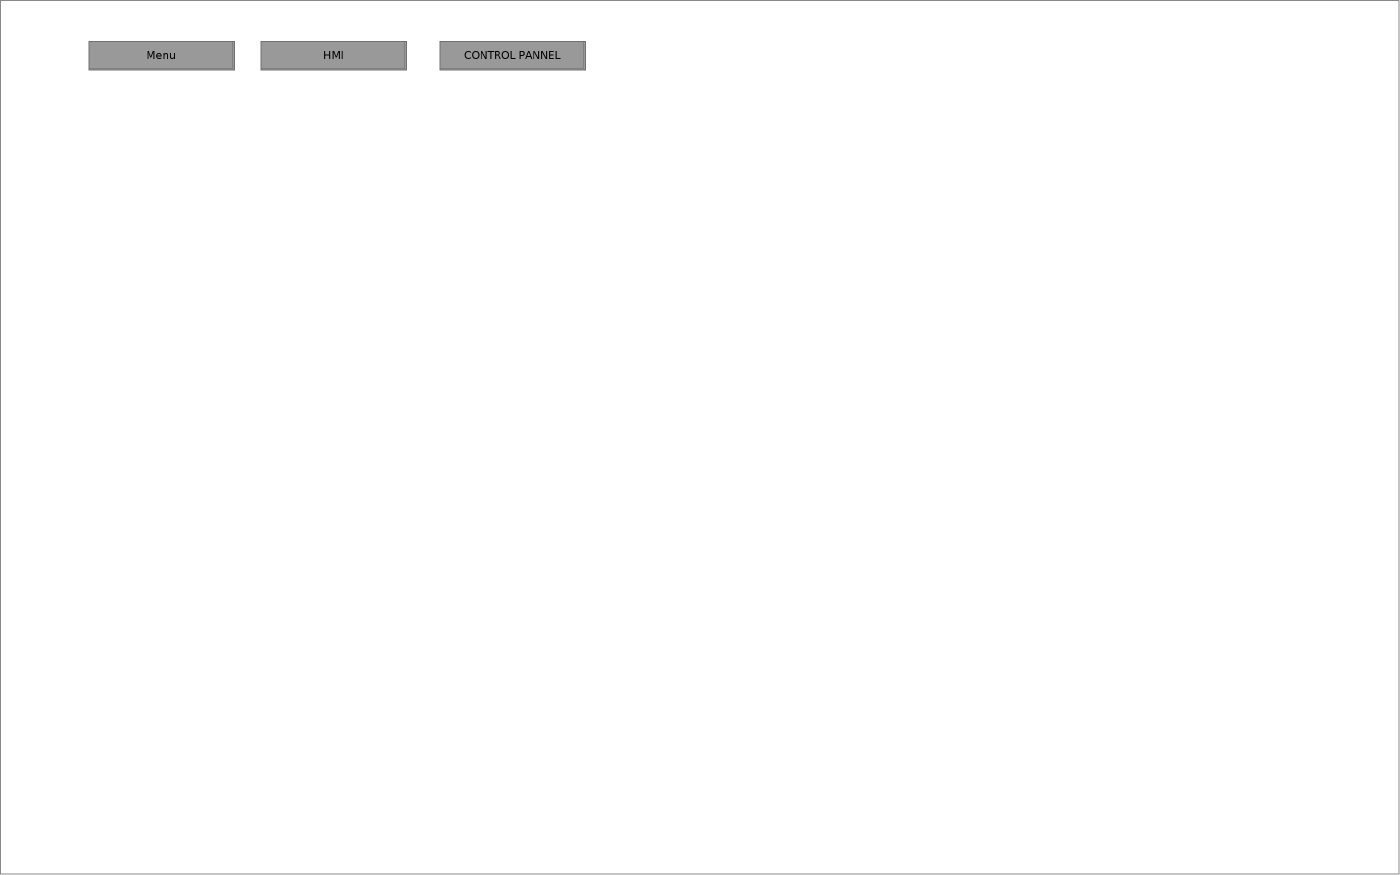
VISUALIZATION Menu  // 1440x900
    Button (91,42 150x30), "Menu"
        OnMouseClick: change screen: Menu
    Button (268,42 150x30), "HMI"
        OnMouseClick: change screen: Visualization
    Button (452,42 150x30), "CONTROL PANNEL"
        OnMouseClick: change screen: Pannello_Controllo
END_VISUALIZATION

(* stored: Version 1.1.0.1
   Visu Menu: Id {7320c326-8624-48f7-a2f5-9547eeaab468} *)
